FUNCTION_BLOCK LOG_W (* Composite FB wrapping other FBs *)
  (* Standard: 61499-2 *)
  (* Version 1.0, 2021-08-05, dorofeev *)
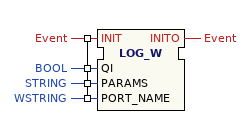
  EVENT_INPUT
    INIT WITH PORT_NAME, PARAMS, QI; (* Initialization Request *)
  END_EVENT
  EVENT_OUTPUT
    INITO;
  END_EVENT
  VAR_INPUT
    QI : BOOL; (* Input event qualifier *)
    PARAMS : STRING;
    PORT_NAME : WSTRING;
  END_VAR
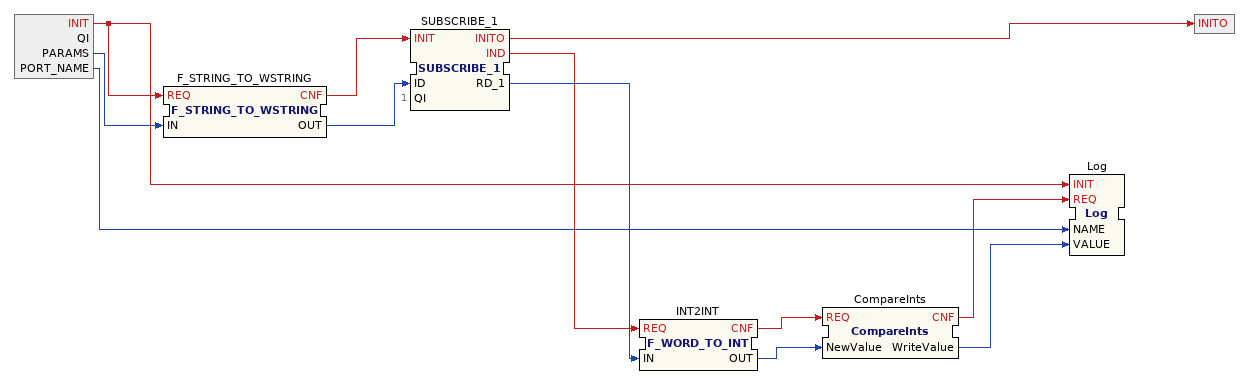
  FBS
    F_STRING_TO_WSTRING : F_STRING_TO_WSTRING;
    SUBSCRIBE_1 : SUBSCRIBE_1(QI := 1);
    Log : Log;
    INT2INT : F_WORD_TO_INT;
    CompareInts : CompareInts;
  END_FBS
  EVENT_CONNECTIONS
    INIT TO F_STRING_TO_WSTRING.REQ;
    F_STRING_TO_WSTRING.CNF TO SUBSCRIBE_1.INIT;
    SUBSCRIBE_1.INITO TO INITO;
    SUBSCRIBE_1.IND TO INT2INT.REQ;
    INT2INT.CNF TO CompareInts.REQ;
    CompareInts.CNF TO Log.REQ;
    INIT TO Log.INIT;
  END_CONNECTIONS
  DATA_CONNECTIONS
    PARAMS TO F_STRING_TO_WSTRING.IN;
    F_STRING_TO_WSTRING.OUT TO SUBSCRIBE_1.ID;
    PORT_NAME TO Log.NAME;
    SUBSCRIBE_1.RD_1 TO INT2INT.IN;
    INT2INT.OUT TO CompareInts.NewValue;
    CompareInts.WriteValue TO Log.VALUE;
  END_CONNECTIONS
END_FUNCTION_BLOCK
